FUNCTION_BLOCK INTERNAL FB_ActionTestObject EXTENDS FB_Object IMPLEMENTS I_CyclicTask
VAR
    _nCounter: UDINT;
    _bActivated: BOOL;
END_VAR

METHOD Activate
VAR_INPUT
    bActivate: BOOL;
END_VAR
THIS^._bActivated := bActivate;
END_METHOD

PROPERTY bIsActivated : BOOL
GET
bIsActivated := THIS^._bActivated;
END_GET
END_PROPERTY

PROPERTY nCounter : UDINT
GET
nCounter := THIS^._nCounter;
END_GET
END_PROPERTY

METHOD Run
VAR_INPUT
END_VAR
THIS^._nCounter := THIS^._nCounter + 1;
END_METHOD

END_FUNCTION_BLOCK

(* stored: Version 1.1.0.1, ProductVersion 3.1.4024.12
   POU FB_ActionTestObject: Id {5641797a-cb27-04c1-000a-970c08e21dc3}, SpecialFunc None
   Method Activate: Id {2b889140-d7a5-0a56-3b9c-f3ac573149f1}
   Property bIsActivated: Id {3e7170b5-2443-0894-1fb8-43b92a28c90a}
   Get Get: Id {f428bd93-865d-0a37-24d5-d5d1f2822df6}
   Property nCounter: Id {70dcdeac-c026-025c-024e-45088ae711f9}
   Get Get: Id {c78e7ebd-d2c8-03ed-22d2-b2e81e97bb85}
   Method Run: Id {d54a1ad8-a015-0eed-3045-bd40456160d4} *)
